TYPE (* a Struct holding 2x2 Object IDs *)
  (* Version 1.0, 2026-05-28, franz *)
  PACKAGE isobus::UT::Q::types;
  IMPORT eclipse4diac::core::TypeHash;
  IMPORT isobus::UT::Q::const::IDs::ID_NULL;
  s2x2ObjectIDs : STRUCT
    up : isobus::UT::Q::types::s2ObjectIDs := (u16ObjId := ID_NULL, u16ObjIdA := ID_NULL); (* forward, up, right, clockwise *)
    down : isobus::UT::Q::types::s2ObjectIDs := (u16ObjId := ID_NULL, u16ObjIdA := ID_NULL); (* backward, down, left, counter-clockwise *)
  END_STRUCT;
END_TYPE
